TYPE E_CircuitBreakerControlMode :
(
    MANUAL := 0,        // Manuel kontrol
    AUTO := 1,          // Otomatik kontrol
    REMOTE := 2         // Uzaktan kontrol
);
END_TYPE

(* stored: Version 1.1.0.1, ProductVersion 3.1.4024.15
   EnumerationTextList E_CircuitBreakerControlMode: Id {d54749a8-ce42-48a1-9c45-60611184b3a6} *)
